FUNCTION_BLOCK FB_STATION
VAR_INPUT
	eSTATE:E_STATE:=E_STATE.uninit;
	sSTATION_STATE:STRING:='UNINIT';
	sName:STRING;
	bHOMED : BOOL:=FALSE;
	tACTION:TON;
	bPAUSE:BOOL:=FALSE;
	bHOME: BOOL:=FALSE;
	
	
END_VAR
VAR_OUTPUT
END_VAR
VAR
	bERROR:BOOL;
	bRESET:BOOL;
	bSTART:BOOL:=FALSE;
	iSTATION_STATE:INT:=98;;
	bFIRST_RUN:BOOL:=FALSE;
END_VAR

ACTION aHOME:
bHOME:=TRUE;
END_ACTION

ACTION aRESET:
bRESET:=TRUE;
END_ACTION

ACTION aSTART:
bSTART:=TRUE;
END_ACTION

END_FUNCTION_BLOCK

(* stored: Version 1.1.0.1, ProductVersion 3.1.4024.12
   POU FB_STATION: Id {af24db28-040e-471c-ad69-35306a54a2e6}, SpecialFunc None
   Action aHOME: Id {aa4b3268-468b-451c-a4a6-4f989c2f669f}
   Action aRESET: Id {493c17cd-846f-4d67-8b2d-ec5af866b7f6}
   Action aSTART: Id {3d8a0d55-b032-4923-96f9-b912755fdb9d} *)
